ABB RobotStudio station: Solution6_20230623-195207.rsstn

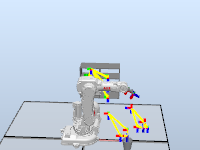
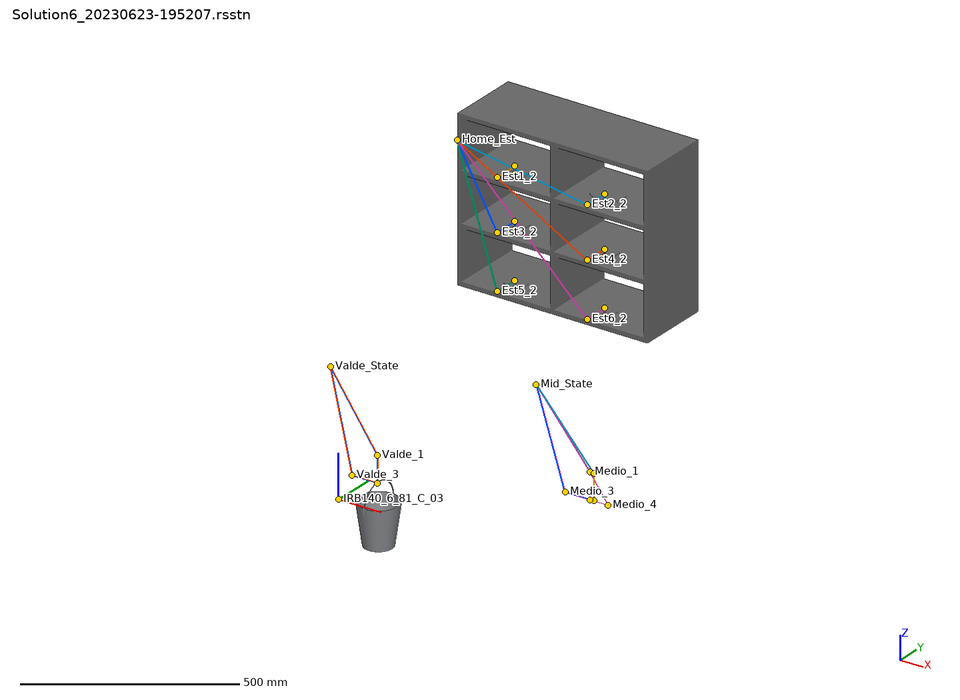
[picture v1: parts stored in the station drawn from their meshes, with robot base, taught points and paths (robot models come from the ABB library and are not in the file)]
Station Solution5 (saved by RobotStudio 22.1.9826.0)
Controller IRB140_6_81
  mechanical unit ROB_1: IRB140_6_81_C_03, 6 joints, base frame (0, 0, 0) mm
Layout (positions relative to the parent item):
  - IRB140_6_81_C_03 [mechanism, from Robots\IRB140_6_81_C_G_03.rslib] at (0, 0, 0) mm; joint values [0, 0, 0, 0, 0.5236, 0] (rad or m)
  - Balde [part] at (450, -500, 250) mm, rotated rx 90 ry 0 rz 0 deg, size 106 x 161 x 120.5 mm
  - tool5 [mechanism] at (506.29, 0, 679.5) mm, rotated rx 180 ry 60 rz 180 deg
      TCP gancho at (0, 73, 40) mm, rotated rx -90 ry 0 rz 0 deg
      TCP ventosa at (22.5, 86.25, -35) mm, rotated rx -90 ry 0 rz -90 deg
      links: herramienta5
  - Estanteria2 [part] at (300, 650, 340) mm, rotated rx 90 ry 0 rz -90 deg, size 200 x 436 x 528 mm
Attachment: tool5 is attached to IRB140_6_81_C_03 / Link6
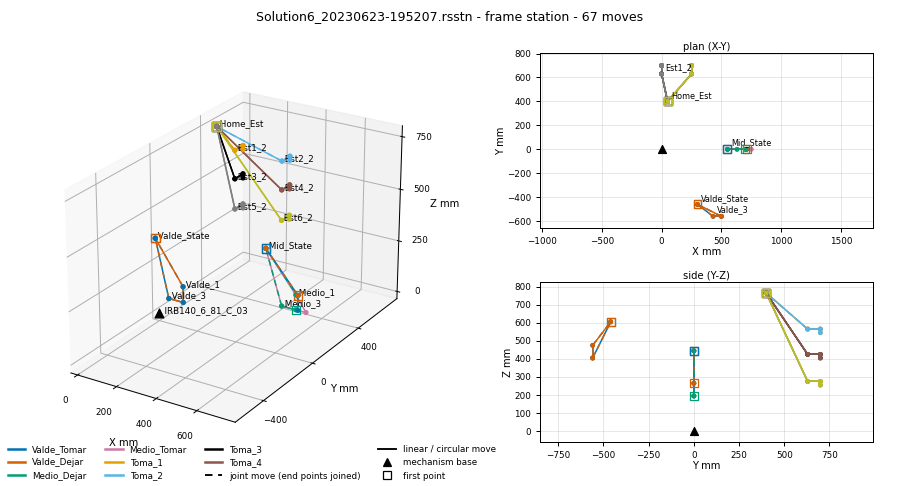
[picture p0: tool path of Solution6_20230623-195207.rsstn in frame station, 67 of 68 moves have a stored position in this frame; points joined in program order, loops and branches not executed]
Targets, tools, work objects and paths stored in the station, written as RAPID:
! task T_ROB1
MODULE CalibData
  TASK PERS wobjdata Mid:=[FALSE,TRUE,"",[[700,0,195],[0,0,1,0]],[[0,0,0],[1,0,0,0]]];
  TASK PERS wobjdata Estanteria:=[FALSE,TRUE,"",[[0,700,565],[0,-0.707106781,0.707106781,0]],[[0,0,0],[1,0,0,0]]];
  TASK PERS wobjdata Vald:=[FALSE,TRUE,"",[[500,-560,405],[0,0,1,0]],[[0,0,0],[1,0,0,0]]];
  PERS tooldata gancho:=[TRUE,[[0,-40,73],[1,0,0,0]],[1,[0,0,1],[1,0,0,0],0,0,0]];
  PERS tooldata ventosa:=[TRUE,[[22.5,35,86.245],[0.707106781,0,0.707106781,0]],[1,[0,0,1],[1,0,0,0],0,0,0]];
ENDMODULE

! task T_ROB1
MODULE Module1
  CONST robtarget Medio_2:=[[0,0,0],[1,0,0,0],[0,0,0,0],[9E+09,9E+09,9E+09,9E+09,9E+09,9E+09]];
  CONST robtarget Medio_1:=[[0,0,-70],[1,0,0,0],[0,0,0,0],[9E+09,9E+09,9E+09,9E+09,9E+09,9E+09]];
  CONST robtarget Medio_3:=[[70,0,0],[1,0,0,0],[0,0,0,0],[9E+09,9E+09,9E+09,9E+09,9E+09,9E+09]];
  CONST robtarget Mid_State:=[[150,0,-250],[1,0,0,0],[0,0,0,0],[9E+09,9E+09,9E+09,9E+09,9E+09,9E+09]];
  CONST robtarget Est1:=[[0,0,0],[1,0,0,0],[0,-1,0,1],[9E+09,9E+09,9E+09,9E+09,9E+09,9E+09]];
  CONST robtarget Est2:=[[0,-250,0],[1,0,0,0],[0,-1,0,1],[9E+09,9E+09,9E+09,9E+09,9E+09,9E+09]];
  CONST robtarget Est4:=[[0,-250,140],[1,0,0,0],[0,-1,0,1],[9E+09,9E+09,9E+09,9E+09,9E+09,9E+09]];
  CONST robtarget Est3:=[[0,0,140],[1,0,0,0],[0,-1,0,1],[9E+09,9E+09,9E+09,9E+09,9E+09,9E+09]];
  CONST robtarget Est5:=[[0,0,290],[1,0,0,0],[0,-1,0,1],[9E+09,9E+09,9E+09,9E+09,9E+09,9E+09]];
  CONST robtarget Est6:=[[0,-250,290],[1,0,0,0],[0,-1,0,1],[9E+09,9E+09,9E+09,9E+09,9E+09,9E+09]];
  CONST robtarget Est1_2:=[[70,0,0],[1,0,0,0],[0,-1,0,1],[9E+09,9E+09,9E+09,9E+09,9E+09,9E+09]];
  CONST robtarget Est2_2:=[[70,-250,0],[1,0,0,0],[0,-1,0,1],[9E+09,9E+09,9E+09,9E+09,9E+09,9E+09]];
  CONST robtarget Est3_2:=[[70,0,140],[1,0,0,0],[0,-1,0,1],[9E+09,9E+09,9E+09,9E+09,9E+09,9E+09]];
  CONST robtarget Est4_2:=[[70,-250,140],[1,0,0,0],[0,-1,0,1],[9E+09,9E+09,9E+09,9E+09,9E+09,9E+09]];
  CONST robtarget Est5_2:=[[70,0,290],[1,0,0,0],[0,0,1,1],[9E+09,9E+09,9E+09,9E+09,9E+09,9E+09]];
  CONST robtarget Est6_2:=[[70,-250,290],[1,0,0,0],[0,-1,0,1],[9E+09,9E+09,9E+09,9E+09,9E+09,9E+09]];
  CONST robtarget Home_Est:=[[300,-50,-200],[1,0,0,0],[0,-1,0,1],[9E+09,9E+09,9E+09,9E+09,9E+09,9E+09]];
  CONST robtarget Valde_2:=[[0,0,0],[1,0,0,0],[-1,0,-1,0],[9E+09,9E+09,9E+09,9E+09,9E+09,9E+09]];
  CONST robtarget Valde_1:=[[0,0,-70],[1,0,0,0],[-1,0,-1,0],[9E+09,9E+09,9E+09,9E+09,9E+09,9E+09]];
  CONST robtarget Valde_3:=[[70,0,0],[1,0,0,0],[-1,0,-1,0],[9E+09,9E+09,9E+09,9E+09,9E+09,9E+09]];
  CONST robtarget Valde_State:=[[200,100,-200],[1,0,0,0],[0,0,0,0],[9E+09,9E+09,9E+09,9E+09,9E+09,9E+09]];
  CONST robtarget Est1_3:=[[0,0,20],[1,0,0,0],[0,-1,0,1],[9E+09,9E+09,9E+09,9E+09,9E+09,9E+09]];
  CONST robtarget Est2_3:=[[0,-250,20],[1,0,0,0],[0,-1,0,1],[9E+09,9E+09,9E+09,9E+09,9E+09,9E+09]];
  CONST robtarget Est3_3:=[[0,0,160],[1,0,0,0],[0,-1,0,1],[9E+09,9E+09,9E+09,9E+09,9E+09,9E+09]];
  CONST robtarget Est4_3:=[[0,-250,160],[1,0,0,0],[0,-1,0,1],[9E+09,9E+09,9E+09,9E+09,9E+09,9E+09]];
  CONST robtarget Est5_3:=[[0,0,310],[1,0,0,0],[0,-1,0,1],[9E+09,9E+09,9E+09,9E+09,9E+09,9E+09]];
  CONST robtarget Est6_3:=[[0,-250,310],[1,0,0,0],[0,-1,0,1],[9E+09,9E+09,9E+09,9E+09,9E+09,9E+09]];
  CONST robtarget Soltar_2:=[[-10,0,-70],[0.707106781,0,0.707106781,0],[0,0,0,0],[9E+09,9E+09,9E+09,9E+09,9E+09,9E+09]];
  CONST robtarget Soltar_1:=[[-10,0,0],[0.707106781,0,0.707106781,0],[0,0,0,0],[9E+09,9E+09,9E+09,9E+09,9E+09,9E+09]];
  CONST robtarget Soltar_State:=[[150,0,-250],[0.707106781,0,0.707106781,0],[-1,0,-1,0],[9E+09,9E+09,9E+09,9E+09,9E+09,9E+09]];
  CONST robtarget Medio_4:=[[-50,0,0],[1,0,0,0],[0,0,0,0],[9E+09,9E+09,9E+09,9E+09,9E+09,9E+09]];
  CONST jointtarget JointTarget_1:=[[0,0,0,0,30,0],[9E+09,9E+09,9E+09,9E+09,9E+09,9E+09]];
  PROC Valde_Tomar()
    MoveJ Valde_State,v600,z100,gancho\WObj:=Vald;
    MoveL Valde_3,v200,z100,gancho\WObj:=Vald;
    MoveL Valde_2,v200,z100,gancho\WObj:=Vald;
    MoveL Valde_1,v100,z100,gancho\WObj:=Vald;
    MoveJ Valde_State,v50,z100,gancho\WObj:=Vald;
  ENDPROC
  PROC Valde_Dejar()
    MoveJ Valde_State,v600,z100,gancho\WObj:=Vald;
    MoveL Valde_1,v200,z100,gancho\WObj:=Vald;
    MoveL Valde_2,v200,z100,gancho\WObj:=Vald;
    MoveL Valde_3,v200,z100,gancho\WObj:=Vald;
    MoveJ Valde_State,v1000,z100,gancho\WObj:=Vald;
  ENDPROC
  PROC Medio_Dejar()
    MoveJ Mid_State,v100,z100,gancho\WObj:=Mid;
    MoveL Medio_1,v50,z10,gancho\WObj:=Mid;
  ENDPROC
  PROC Medio_Tomar()
    MoveJ Mid_State,v1000,z100,gancho\WObj:=Mid;
    MoveL Medio_3,v200,z100,gancho\WObj:=Mid;
    MoveL Medio_4,v200,z100,gancho\WObj:=Mid;
    MoveL Medio_1,v200,z100,gancho\WObj:=Mid;
    MoveJ Mid_State,v1000,z100,gancho\WObj:=Mid;
  ENDPROC
  PROC Toma_1()
    MoveJ Home_Est,v500,z50,ventosa\WObj:=Estanteria;
    MoveL Est1_2,v200,z100,ventosa\WObj:=Estanteria;
    MoveL Est1,v200,z100,ventosa\WObj:=Estanteria;
    MoveL Est1_3,v200,z100,ventosa\WObj:=Estanteria;
    MoveL Est1,v200,z100,ventosa\WObj:=Estanteria;
    MoveL Est1_2,v200,z100,ventosa\WObj:=Estanteria;
    MoveJ Home_Est,v500,z50,ventosa\WObj:=Estanteria;
  ENDPROC
  PROC Toma_2()
    MoveJ Home_Est,v500,z50,ventosa\WObj:=Estanteria;
    MoveL Est2_2,v200,z100,ventosa\WObj:=Estanteria;
    MoveL Est2,v200,z100,ventosa\WObj:=Estanteria;
    MoveL Est2_3,v200,z100,ventosa\WObj:=Estanteria;
    MoveL Est2,v200,z100,ventosa\WObj:=Estanteria;
    MoveL Est2_2,v200,z100,ventosa\WObj:=Estanteria;
    MoveJ Home_Est,v500,z50,ventosa\WObj:=Estanteria;
  ENDPROC
  PROC Toma_3()
    MoveJ Home_Est,v500,z50,ventosa\WObj:=Estanteria;
    MoveL Est3_2,v200,z100,ventosa\WObj:=Estanteria;
    MoveL Est3,v200,z100,ventosa\WObj:=Estanteria;
    MoveL Est3_3,v200,z100,ventosa\WObj:=Estanteria;
    MoveL Est3,v200,z100,ventosa\WObj:=Estanteria;
    MoveL Est3_2,v200,z100,ventosa\WObj:=Estanteria;
    MoveL Home_Est,v500,z100,ventosa\WObj:=Estanteria;
  ENDPROC
  PROC Toma_4()
    MoveJ Home_Est,v500,z50,ventosa\WObj:=Estanteria;
    MoveL Est4_2,v200,z100,ventosa\WObj:=Estanteria;
    MoveL Est4,v200,z100,ventosa\WObj:=Estanteria;
    MoveL Est4_3,v200,z100,ventosa\WObj:=Estanteria;
    MoveL Est4,v200,z100,ventosa\WObj:=Estanteria;
    MoveL Est4_2,v200,z100,ventosa\WObj:=Estanteria;
    MoveL Home_Est,v500,z100,ventosa\WObj:=Estanteria;
  ENDPROC
  PROC Toma_5()
    MoveJ Home_Est,v500,z50,ventosa\WObj:=Estanteria;
    MoveL Est5_2,v200,z100,ventosa\WObj:=Estanteria;
    MoveL Est5,v200,z100,ventosa\WObj:=Estanteria;
    MoveL Est5_3,v200,z100,ventosa\WObj:=Estanteria;
    MoveL Est5,v200,z100,ventosa\WObj:=Estanteria;
    MoveL Est5_2,v200,z100,ventosa\WObj:=Estanteria;
    MoveL Home_Est,v500,z100,ventosa\WObj:=Estanteria;
  ENDPROC
  PROC Toma_6()
    MoveJ Home_Est,v500,z50,ventosa\WObj:=Estanteria;
    MoveL Est6_2,v200,z100,ventosa\WObj:=Estanteria;
    MoveL Est6,v200,z100,ventosa\WObj:=Estanteria;
    MoveL Est6_3,v200,z100,ventosa\WObj:=Estanteria;
    MoveL Est6,v200,z100,ventosa\WObj:=Estanteria;
    MoveL Est6_2,v200,z100,ventosa\WObj:=Estanteria;
    MoveL Home_Est,v500,z100,ventosa\WObj:=Estanteria;
  ENDPROC
  PROC Soltar_Ficha()
    MoveJ Soltar_State,v400,z100,ventosa\WObj:=Mid;
    MoveL Soltar_2,v200,z100,ventosa\WObj:=Mid;
    MoveL Soltar_1,v200,z100,ventosa\WObj:=Mid;
  ENDPROC
  PROC Soltar_Volver()
    MoveL Soltar_2,v200,z100,ventosa\WObj:=Mid;
    MoveJ Soltar_State,v600,z100,ventosa\WObj:=Mid;
  ENDPROC
  PROC Medio_Dejar2()
    MoveL Medio_2,v20,z10,gancho\WObj:=Mid;
    MoveL Medio_3,v50,z100,gancho\WObj:=Mid;
    MoveJ Mid_State,v1000,z100,gancho\WObj:=Mid;
  ENDPROC
  PROC GoHome()
    MoveAbsJ JointTarget_1,v500,z100,tool0\WObj:=Mid;
  ENDPROC
ENDMODULE

